FUNCTION_BLOCK FB_ExhAirModbus
VAR_INPUT
	nSet	:	WORD;	//Setpoint in hundreds of a percent
END_VAR
VAR_OUTPUT
	nAct	:	Array[11..12] of WORD;	//Actual volume flow in m^3/h
END_VAR
VAR
	Step	:	INT		:=	1;
	ModAdr	:	BYTE	:=	11;
	
	nZwang	:	WORD;
	bZwang	:	BOOL	:=	FALSE;
	
	fbModK6		:	ModbusRtuMaster_KL6x22B;
	bModErr		:	BOOL;
	ErrID		:	MODBUS_ERRORS;
END_VAR

CASE Step OF
	
	1:	//start writing setpoint to nozzle
		IF nSet = 65535 THEN
			Step	:=	20;	//Control override
			bZwang	:=	TRUE;
		ELSE
			IF bZwang THEN
				Step :=	30;
			ELSE
				fbModK6.WriteSingleRegister(
						UnitID		:=	ModAdr,	//Modbus address of slave
						MBAddr		:=	0,	//Register address
						Quantity	:=	1,	//Number of registers to be written
						pMemoryAddr	:=	ADR(nSet),		//Pointer to write data
						cbLength	:=	SIZEOF(nSet),	//Size of write data
						Timeout		:=	T#5S,			//Time to wait for the slave to respond
						Execute		:=	TRUE
					);
					Step	:=	2;
			END_IF
		END_IF
		
	2:	//finish writing process
		fbModK6.WriteSingleRegister(Execute:=FALSE, Error=>bModErr, ErrorID=>ErrID);
		IF NOT fbModK6.BUSY THEN
			Step	:=	3;	//go to next step when writing process has finished
		END_IF
		IF fbModK6.Error THEN
			Step	:=	99;
		END_IF
		
	3:	//start reading volume flow
		fbModK6.ReadRegs(
			UnitID		:=	ModAdr,	//Modbus address of slave
			MBAddr		:=	7,	//Register address
			Quantity	:=	1,	//Number of registers to be read
			pMemoryAddr	:=	ADR(nAct[ModAdr]),		//Pointer to read data
			cbLength	:=	SIZEOF(nAct[ModAdr]),	//Size of read data
			Timeout		:=	T#5S,			//Time to wait for the slave to respond
			Execute		:=	TRUE
		);
		Step	:=	4;
		
	4:	//finish reading process
		fbModK6.ReadRegs(Execute:=FALSE, Error=>bModErr, ErrorID=>ErrID);
		IF NOT fbModK6.BUSY THEN
			Step	:=	5;	//go to next step when reading process has finished
		END_IF
		IF fbModK6.Error THEN
			Step	:=	99;
		END_IF
		
	5:	//go to next nozzle or finish operation
		ModAdr	:=	ModAdr+1;
		IF ModAdr <= 12 THEN
			Step	:=	1;	//start process for other actuator
		ELSE
			Step	:=	6;
		END_IF
		
	6:	//prepare next operation
		ModAdr	:=	11;
		Step	:=	1;
		
	20: //Activate control override for actuator 1
		nZwang	:=	2;
		fbModK6.WriteSingleRegister(
			UnitID		:=	11,	//Modbus address of slave
			MBAddr		:=	1,	//Regster address
			Quantity	:=	1,	//Number of registers to be written
			pMemoryAddr	:=	ADR(nZwang),		//Pointer to write data
			cbLength	:=	SIZEOF(nZwang),	//Size of write data
			Timeout		:=	T#5S,				//Time to wait for the slave to respond
			Execute		:=	TRUE
		);
		Step	:=	21;
	
	21:	//finish writing process
		fbModK6.WriteSingleRegister(Execute:=FALSE, Error=>bModErr, ErrorID=>ErrID);
		IF NOT fbModK6.BUSY THEN
			Step	:=	22;	//go to next step when writing process has finished
		END_IF
		IF fbModK6.Error THEN
			Step	:=	99;
		END_IF
		
	22: //Activate control override for actuator 2		
		nZwang	:=	2;
		fbModK6.WriteSingleRegister(
			UnitID		:=	12,	//Modbus address of slave
			MBAddr		:=	1,	//Regster address
			Quantity	:=	1,	//Number of registers to be written
			pMemoryAddr	:=	ADR(nZwang),		//Pointer to write data
			cbLength	:=	SIZEOF(nZwang),	//Size of write data
			Timeout		:=	T#5S,				//Time to wait for the slave to respond
			Execute		:=	TRUE
		);
		Step	:=	23;
	
	23:	//finish writing process
		fbModK6.WriteSingleRegister(Execute:=FALSE, Error=>bModErr, ErrorID=>ErrID);
		IF NOT fbModK6.BUSY THEN
			Step	:=	3;	//go to next step when writing process has finished
		END_IF
		IF fbModK6.Error THEN
			Step	:=	99;
		END_IF
		
	30: //End control override for actuator 1
		nZwang	:=	0;
		fbModK6.WriteSingleRegister(
			UnitID		:=	11,	//Modbus address of slave
			MBAddr		:=	1,	//Register address
			Quantity	:=	1,	//Number of registers to be written
			pMemoryAddr	:=	ADR(nZwang),		//Pointer to write data
			cbLength	:=	SIZEOF(nZwang),	//Size of write data
			Timeout		:=	T#5S,				//Time to wait for the slave to respond
			Execute		:=	TRUE
		);
		Step	:=	31;
	
	31:	//finish writing process
		fbModK6.WriteSingleRegister(Execute:=FALSE, Error=>bModErr, ErrorID=>ErrID);
		IF NOT fbModK6.BUSY THEN
			bZwang	:=	FALSE;
			Step	:=	32;
		END_IF
		IF fbModK6.Error THEN
			Step	:=	99;
		END_IF
		
	32: //End control override for actuator 2
		nZwang	:=	0;
		fbModK6.WriteSingleRegister(
			UnitID		:=	12,	//Modbus address of slave
			MBAddr		:=	1,	//Register address
			Quantity	:=	1,	//Number of registers to be written
			pMemoryAddr	:=	ADR(nZwang),		//Pointer to write data
			cbLength	:=	SIZEOF(nZwang),	//Size of write data
			Timeout		:=	T#5S,				//Time to wait for the slave to respond
			Execute		:=	TRUE
		);
		Step	:=	33;
	
	33:	//finish writing process
		fbModK6.WriteSingleRegister(Execute:=FALSE, Error=>bModErr, ErrorID=>ErrID);
		IF NOT fbModK6.BUSY THEN
			bZwang	:=	FALSE;
			Step	:=	1;	//start normal writing process
		END_IF
		IF fbModK6.Error THEN
			Step	:=	99;
		END_IF
				
	99:	//Error
		
END_CASE

END_FUNCTION_BLOCK

(* stored: Version 1.1.0.1, ProductVersion 3.1.4022.10
   POU FB_ExhAirModbus: Id {a1f22dcb-b8fd-44f1-a25d-afe2803e67d0}, SpecialFunc None *)
